PROGRAM JIG001_VOLVOL125
VAR
END_VAR

END_PROGRAM

(* stored: Version 1.1.0.1, ProductVersion 3.1.4022.18
   POU JIG001_VOLVOL125: Id {c550c97b-b259-4297-8015-22414febe0a6}, SpecialFunc None *)
